// TIA Portal V21 export
VAR_GLOBAL   // PLC tag table "K_Valvola"
END_VAR
VAR_GLOBAL CONSTANT   // user constants
   K_Valvola_A : Int := 1;
   K_Valvola_A1 : Int := 2;
   K_Valvola_B : Int := 3;
   K_Valvola_B1 : Int := 4;
   K_Valvola_C : Int := 5;
   K_Valvola_D : Int := 6;
   K_Valvola_D1 : Int := 7;
   K_Valvola_D2 : Int := 8;
   K_Valvola_E : Int := 9;
   K_Valvola_E1 : Int := 10;
   K_Valvola_F : Int := 11;
   K_Valvola_G : Int := 12;
   K_Valvola_H : Int := 13;
   K_Valvola_H1 : Int := 14;
   K_Valvola_I : Int := 15;
   K_Valvola_L : Int := 16;
   K_Valvola_N : Int := 17;
   K_Valvola_N1 : Int := 18;
   K_Valvola_R : Int := 19;
   K_Valvola_U : Int := 20;
   K_Valvola_UU : Int := 21;
   K_Valvola_V : Int := 22;
   K_Valvola_VV : Int := 23;
   K_Valvola_UV : Int := 24;
   K_Valvola_Z : Int := 25;
   K_Valvola_Z1 : Int := 26;
   K_Valvola_Y : Int := 27;
   K_Valvola_Y1 : Int := 28;
   K_Valvola_Y2 : Int := 29;
   K_Valvola_J : Int := 30;
   K_Valvola_X : Int := 31;
   K_Valvola_XXX : Int := 32;
   K_Valvola_XX : Int := 33;
   K_Valvola_CP1 : Int := 34;
   K_Valvola_CP2 : Int := 35;
   K_Valvola_CP3 : Int := 36;
   K_Valvola_EV103_6 : Int := 37;
   K_Valvola_X2 : Int := 38;
END_VAR
